RoboDK station: ur20_proyecto_final.rdk

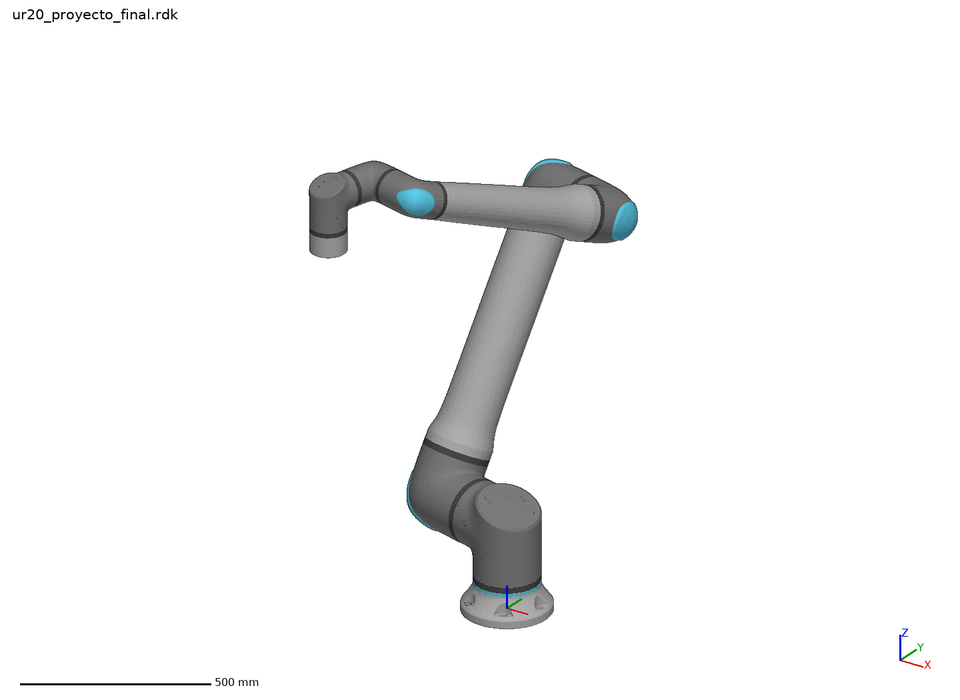
[picture v0: the station drawn from its stored meshes, robots at their saved joint values, targets as dots, program paths as lines]
Station ur20_proyecto_final (saved by RoboDK 5.9.4). Poses are relative to the parent item; angles as X-Y-Z fixed-axis rotations.
  - frame UR20 Base at (0, 0, 0) mm
    - robot UR20: 6 axes
        modified DH rows (alpha deg, a mm, theta deg, d mm): 0, 0, 0, 236.2; 90, 0, -180, 0; 0, 861.8, 0, 0; 0, 727.7, 0, 201.9; -90, 0, 0, 159.4; 90, 0, 180, 154.8
        joint limits [-360, -360, -360, -360, -360, -360] to [360, 360, 360, 360, 360, 360]; home [0, -90, -90, 0, 90, 0]; saved at [-103.65, -63.01, -95.58, 248.5, 90, -166.23]
